TYPE ST_HeatStakeProcessSettings :
STRUCT
    tContactTime     : TIME := T#3S;
    rDownPressureBar : LREAL := 0.5;
END_STRUCT
END_TYPE

(* stored: Version 1.1.0.1, ProductVersion 3.1.4026.18
   DUT ST_HeatStakeProcessSettings: Id {16deca7e-e66f-4e33-94b5-04afad4e2305} *)
